(* PLC project prj, KAIST_DSLAB noNameNow 1, author bwkim *)
(* stored: creationDateTime 2015-7-21T04:48:50, modificationDateTime 2015-7-21T04:48:50 *)

PROGRAM Program1____FFTD
  VAR
    PTRIP_TON : null;
  END_VAR
  VAR
    TRIP_TON : null;
  END_VAR
  VAR
    VF_PTRIP_TON : null;
  END_VAR
  VAR_INPUT
    PK_DELAY : INT := 100;
  END_VAR
  VAR_INPUT
    K_DELAY : INT := 100;
  END_VAR
  VAR_OUTPUT
    PTON_et : INT;
  END_VAR
  VAR_OUTPUT
    TON_et : INT;
  END_VAR
  VAR_OUTPUT
    PTRIP : BOOL := FALSE;
  END_VAR
  VAR_OUTPUT
    TRIP : BOOL := FALSE;
  END_VAR
  VAR_IN_OUT
    PTRIP_LOGIC : INT;
  END_VAR
  VAR_IN_OUT
    TRIP_LOGIC : INT;
  END_VAR
  VAR_IN_OUT
    HB_t0 : INT;
  END_VAR
  VAR_IN_OUT
    HB_ERR : INT;
  END_VAR
  VAR_IN_OUT
    CTUD_qd : INT;
  END_VAR
  VAR_IN_OUT
    CTUD_qu : INT;
  END_VAR
  VAR_IN_OUT
    HB_ERR_CNT : INT;
  END_VAR
  VAR  (* added by the conversion: wires and edge detectors of the diagram *)
    _SEL_BOOL49_OUT : INT;
    _SEL_BOOL51_OUT : INT;
    _SEL_REAL52_OUT : ANY;
    _AND2_BOOL36_OUT : INT;
    _SEL_REAL50_OUT : ANY;
    _AND2_BOOL38_OUT : INT;
    _AND2_BOOL41_OUT : ANY;
  END_VAR

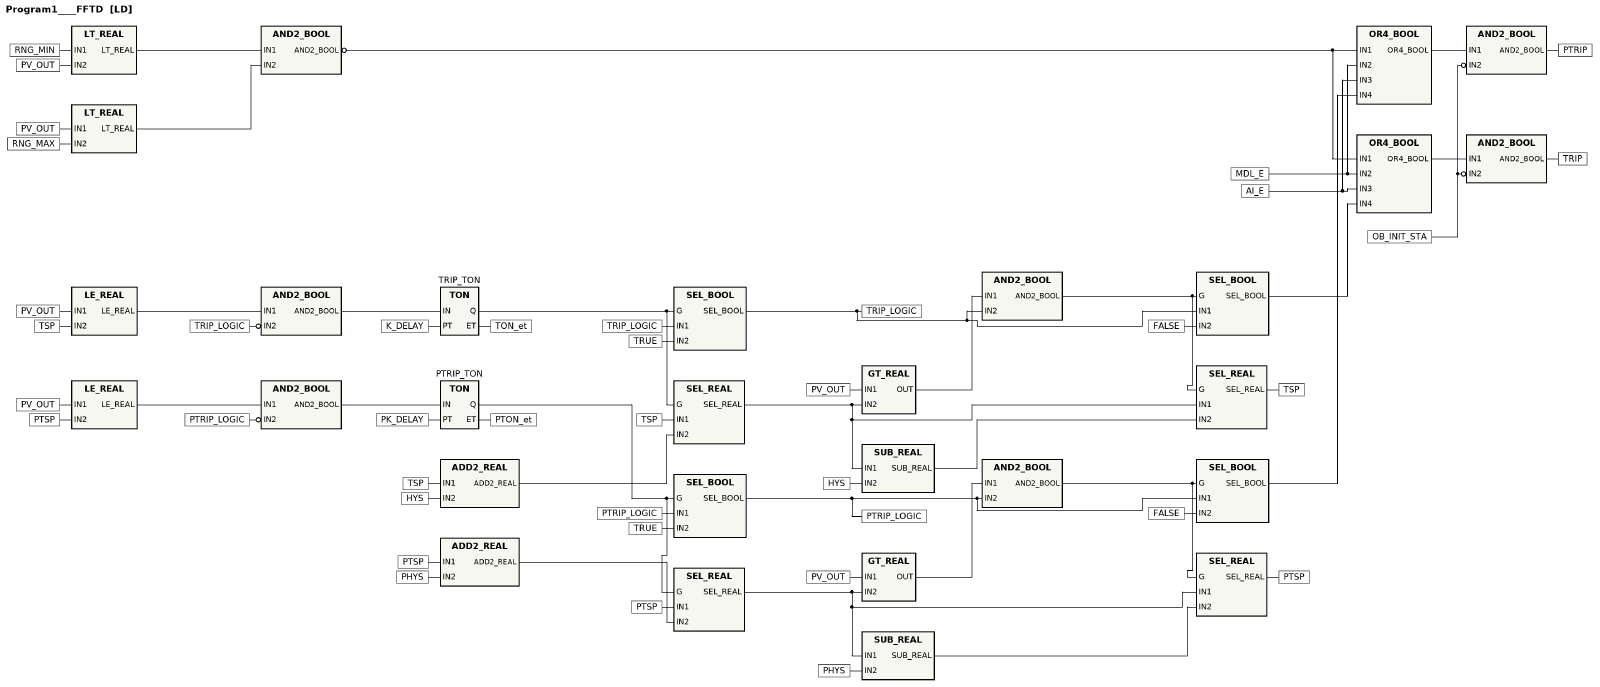
(* LD diagram, written out as Structured Text *)
PTRIP_TON(IN := AND2_BOOL(LE_REAL(PV_OUT, PTSP), NOT PTRIP_LOGIC), PT := PK_DELAY);
_SEL_BOOL49_OUT := SEL_BOOL(PTRIP_TON.Q, PTRIP_LOGIC, TRUE);
PTRIP_LOGIC := _SEL_BOOL49_OUT;
PTON_et := PTRIP_TON.ET;
TRIP_TON(IN := AND2_BOOL(LE_REAL(PV_OUT, TSP), NOT TRIP_LOGIC), PT := K_DELAY);
_SEL_BOOL51_OUT := SEL_BOOL(TRIP_TON.Q, TRIP_LOGIC, TRUE);
TRIP_LOGIC := _SEL_BOOL51_OUT;
TON_et := TRIP_TON.ET;
_SEL_REAL52_OUT := SEL_REAL(TRIP_TON.Q, TSP, ADD2_REAL(TSP, HYS));
_AND2_BOOL36_OUT := AND2_BOOL(GT_REAL(PV_OUT, _SEL_REAL52_OUT), _SEL_BOOL51_OUT);
TSP := SEL_REAL(_AND2_BOOL36_OUT, _SEL_REAL52_OUT, SUB_REAL(_SEL_REAL52_OUT, HYS));
_SEL_REAL50_OUT := SEL_REAL(PTRIP_TON.Q, PTSP, ADD2_REAL(PTSP, PHYS));
_AND2_BOOL38_OUT := AND2_BOOL(GT_REAL(PV_OUT, _SEL_REAL50_OUT), _SEL_BOOL49_OUT);
PTSP := SEL_REAL(_AND2_BOOL38_OUT, _SEL_REAL50_OUT, SUB_REAL(_SEL_REAL50_OUT, PHYS));
_AND2_BOOL41_OUT := AND2_BOOL(LT_REAL(RNG_MIN, PV_OUT), LT_REAL(PV_OUT, RNG_MAX));
PTRIP := AND2_BOOL(OR4_BOOL(_AND2_BOOL41_OUT, MDL_E, AI_E, SEL_BOOL(_AND2_BOOL38_OUT, _SEL_BOOL49_OUT, FALSE)), NOT OB_INIT_STA);
TRIP := AND2_BOOL(OR4_BOOL(_AND2_BOOL41_OUT, MDL_E, AI_E, SEL_BOOL(_AND2_BOOL36_OUT, _SEL_BOOL51_OUT, FALSE)), NOT OB_INIT_STA);
END_PROGRAM
